// LS Electric XG5000 project: CTU
// PLC LSPLC
// module base 0 slot 0: 입출력 모듈:XBC-DR30S (DC 24V 입력 18점, 릴레이 출력 12점)

PROGRAM CTU (task: 스캔 프로그램)

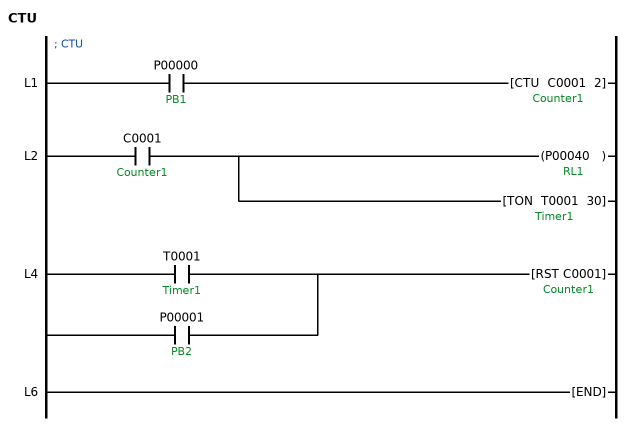
// CTU
; L1
LOAD      P00000	// PB1
CTU       C0001 2	// Counter1
; L2
LOAD      C0001	// Counter1
OUT       P00040	// RL1
TON       T0001 30	// Timer1
; L4
LOAD      T0001	// Timer1
OR        P00001	// PB2
RST       C0001	// Counter1
; L6
END